// TIA Portal V16 export
// export: Created 2022-04-26T19:39:02.1727299Z, ExportSetting WithDefaults, DisplayName Totally Integrated Automation Portal, DisplayVersion V16 Update 1, DisplayName TIA Portal Version Control Interface, DisplayVersion V16, DisplayName TIA Portal Openness, DisplayVersion V16, DisplayName SINAMICS Startdrive Advanced, DisplayVersion V16 Update 5, DisplayName SINAMICS Startdrive G130, G150, S120, S150, SINAMICS MV, S210, DisplayVersion V16 Update 5, DisplayName SINAMICS Startdrive G110M, G120, G120C, G120D, G120P, G115D, DisplayVersion V16 Update 5, DisplayName STEP 7 Professional, DisplayVersion V16, DisplayName STEP 7 Safety, DisplayVersion V16, DisplayName WinCC Advanced, DisplayVersion V16
FUNCTION_BLOCK "FB110 - Scroll Allarmi"   // FB110, LAD
{ S7_Optimized_Access := 'TRUE' }
VERSION : 0.1
// stored: AutoNumber false, IsIECCheckEnabled false, IsRetainMemResEnabled false, MemoryReserve 100, SetENOAutomatically false, UDAEnableTagReadback false
   VAR_INPUT
      "Timer" : Time := T#3S;   // Tempo Per Scroll
      "Numero Di Allarmi" : Int;
   END_VAR
   VAR
      "Timer Scroll" { ExternalAccessible := 'False'; ExternalVisible := 'False'; ExternalWritable := 'False'} : TON_TIME;
      "App.Per Scroll Allarmi" { ExternalAccessible := 'False'; ExternalVisible := 'False'; ExternalWritable := 'False'} : Array[0..80] of Bool;
      "Consenso Timer" { S7_SetPoint := 'True'} : Bool;
      "Uscita Timer" : Bool;
      Cont : Int;
      "App Cont" : Int;
   END_VAR
   VAR_TEMP
      App : Int;
      "By" : Int;   // Byte
      Bt : Int;   // Bit
      "Time Out" : Time;   // Tempo Attuale
   END_VAR
BEGIN

REGION Network 1 (SCL): Copiatura In Array
   // Copio Dalla DB Allarmi Tutti Gli Allarmi sull'Array  "App.Per Scroll Allarmi"

   #App:= 1;
   FOR #By := 0 TO 10 DO
       FOR #Bt := 0 TO 7 DO
           #"App.Per Scroll Allarmi"[#App] := PEEK_BOOL(area := 16#84, dbNumber := 111, byteOffset := 10 + #By, bitOffset := 0 + #Bt);
           #App := #App + 1;
       END_FOR;

   END_FOR;
END_REGION

REGION Network 2 (SCL): Scroll Allarmi
   //Timer Per Scroll
   #"Timer Scroll".TON(IN:=#"Consenso Timer",
                          PT:=#Timer,
                          Q=>#"Uscita Timer",
                          ET=>#"Time Out");


       //IF Reset Timer Alla Fine Del Ciclo
      IF #Cont> 80 & #"App Cont" > 80 THEN
          #Cont:= 0;
          #"App Cont":= 0;
           PRESET_TIMER(PT := T#0s,
                        "TIMER" := #"Timer Scroll");
      END_IF;



      IF #"Uscita Timer" = TRUE THEN
          FOR #Cont:= #"App Cont" TO 80 DO
           IF #"App.Per Scroll Allarmi"[#Cont] = TRUE THEN
               "MainDB".Alm."Numero Allarme Da Visualizzare" := #Cont;
               EXIT;
           END_IF;
           #"App Cont" := 0;
       END_FOR;
       RESET_TIMER(#"Timer Scroll");
       #"App Cont" := #Cont + 1;
   END_IF;
   #"Consenso Timer" := TRUE;
END_REGION
END_FUNCTION_BLOCK
